// TIA Portal V20 export
// export: Created 2026-07-10T11:12:19.8859944Z, ExportSetting WithDefaults, DisplayName Totally Integrated Automation Portal, DisplayVersion V20, DisplayName TIA Portal Openness, DisplayVersion V20, DisplayName TIA Portal Version Control Interface, DisplayVersion V20, DisplayName STEP 7 Professional, DisplayVersion V20, DisplayName STEP 7 Safety, DisplayVersion V20, DisplayName WinCC Basic/Comfort/Advanced, DisplayVersion V20, DisplayName WinCC Unified, DisplayVersion V20
FUNCTION_BLOCK "WaterCounter"   // FB1, SCL
{ S7_Optimized_Access := 'TRUE' }
VERSION : 0.1
// stored: AutoNumber true, IsIECCheckEnabled false, IsRetainMemResEnabled false, MemoryReserve 100, SetENOAutomatically false, UDAEnableTagReadback false
   VAR
      WaterCounter_InWater : "FlowCounter";
      WaterCounter_OutWater : "FlowCounter";
      DelayTON { S7_SetPoint := 'True'} : TON_TIME;
      ChlorCounter_1 { S7_SetPoint := 'True'} : "FlowCounter";
      ChlorCounter_2 { S7_SetPoint := 'True'} : "FlowCounter";
   END_VAR
BEGIN
   #WaterCounter_InWater(Pulse:="WaterCounterInPulse",
                         DailyCount:="MB".Table.WaterCounterIn_DailyCount,
                         TotalCount:="MB".Table.WaterCounterIn_TotalCount,
                         PulseWeight:="MB".Table.WaterCounterInPulseValue,
                         Consumption:="MB".Table.WaterConsumption,
                         DailyValue:="MB".Table.WaterCounterInDailyValue,
                         TotalValue:="MB".Table.WaterCounterInTotalValue);

   #WaterCounter_OutWater(Pulse := "WaterCounterOutPulse",
                          DailyCount := "MB".Table.WaterCounterOut_DailyCount,
                          TotalCount := "MB".Table.WaterCounterOut_TotalCount,
                          PulseWeight := "MB".Table.WaterCounterOut_PulseValue,
                          Consumption := "MB".Table.WaterCounterOut_Consumption,
                          DailyValue := "MB".Table.WaterCounterOut_DailyValue,
                          TotalValue := "MB".Table.WaterCounterOut_TotalValue);

   IF #WaterCounter_OutWater.R_TRIG_Instance.Q THEN
       "Config".WaterPulseDuble := TRUE;
   END_IF;



   IF NOT "MB".Table.Chloration_ChooseCounter THEN
       "ChlorationOut" := "WaterCounterOutPulse";
   ELSE
       "ChlorationOut" := "WaterCounterInPulse";
   END_IF;

   IF "MB".Table.WaterCounterOut_Consumption < 0 THEN
       "FlowAO" := 5520;
   ELSIF "MB".Table.WaterCounterOut_Consumption > 80.0 THEN
       "FlowAO" := 27648;
   ELSE
       "FlowAO" := REAL_TO_INT(("MB".Table.WaterCounterOut_Consumption) / (80) * (27648 - 5520) + 5520);
   END_IF;

   // IF "MB".Table.WaterConsumption < 0 THEN
   //     "OsmosAO" := 5520;
   // ELSIF "MB".Table.WaterConsumption > 80.0 THEN
   //     "OsmosAO" := 27648;
   // ELSE
   //     "OsmosAO" := REAL_TO_INT(("MB".Table.WaterConsumption - "MB".Table.RecerculationFlow) / (80) * (27648 - 5520) + 5520);
   // END_IF;
   // "MB".Table.FlowWithouRecerculation := "MB".Table.WaterConsumption - "MB".Table.RecerculationFlow;
   // IF "MB".Table.FlowWithouRecerculation < 0 THEN
   //     "MB".Table.FlowWithouRecerculation := 0;
   // END_IF;


   #ChlorCounter_1(Pulse:="Doser1",
                   DailyCount:="MB".Table.Doser1_DailyPulses,
                   TotalCount:="MB".Table.Doser1_TotalPulses,
                  PulseWeight:="MB".Table.Doser1_PulseValue,
                  Consumption := "MB".Table.Doser1_Cunsumption,
                  DailyValue:="MB".Table.Doser1_DailyValue,
                  TotalValue:="MB".Table.Doser1_TotalValue);

   #ChlorCounter_2(Pulse := "Doser2",
                   DailyCount := "MB".Table.Doser2_DailyPulses,
                   TotalCount := "MB".Table.Doser2_TotalPulses,
                  PulseWeight := "MB".Table.Doser2_PulseValue,
                  Consumption := "MB".Table.Doser2_Cunsumption,
                  DailyValue := "MB".Table.Doser2_DailyValue,
                  TotalValue := "MB".Table.Doser2_TotalValue);
END_FUNCTION_BLOCK
